# EPICS substitutions: example/example.substitutions
###############################################################################
#
# Positioner template example
#
# $Revision: $
# $Id: $
#
###############################################################################

###############################################################################
#
# Positioner template
#
# The positioner template generates an mbbo record named '$(device):select' that
# is used to select one of n motor positions defined using the position template.
# The output drives the specified motor record '$(motor)'.
#
# interface:
# mbbi   '$(device):select' - use to select the required motor position.
#
# substitutions:
# device  - device name
# motor   - the motor record to be driven
#

file ../db/positioner.template
{
pattern { device, motor }
        { BL18I-DI-PHDGN-01, BL18I-DI-PHDGN-01:MTR }
}

###############################################################################
#
# Position template
# The position template adds '$(device):pos$(idx)' and '$(device):name$(idx)'
# position records to the a positioner template. These specify the motor position
# and the corresponding string name for that position. Up to 16 positions can be
# defined (limited by mbbo record). These records can be changed at run time.
#
# interface
# ao        $(device):pos$(idx)   - use to define the motor position in EGU's at run time
# stringout $(device):name$(idx)  - use to define the name for the position at run time
#
# substitutions:
# device    - device name. This must match the positioner templates $(device) definition.
# pos_name  - the name for the motor position (e.g. a filter name)
# pos_motor - the required motor position in engineering units.
# pos_min   - motor position minimum (in egu's)
# pos_max   - motor position maximum (in egu's)
# pos_egu   - motor position engineering units
# pos_prec  - display precision (PREC) for positions
# idx       - the position suffix (0,1,2...15 corresponding to id)
# id        - one of the EPICS record count prefixes (must be ZR|ON|TW|TH ...FF). (Must be unique for any one positioner)
#

file ../db/position.template
{
pattern { device, pos_name, pos_motor, pos_min, pos_max, pos_egu, pos_prec, idx, id }
        { BL18I-DI-PHDGN-01, filter0, 0, -100, 100, mm, 0, 0, ZR  }
        { BL18I-DI-PHDGN-01, filter1, 20, -100, 100, mm, 0, 1, ON  }
        { BL18I-DI-PHDGN-01, filter2, 50, -100, 100, mm, 0, 2, TW  }
        { BL18I-DI-PHDGN-01, filter3, 95, -100, 100, mm, 0, 3, TH  }
#        { BL18I-DI-PHDGN-01, filter4, 104, -100, 100, mm, 0, 4, FR  }
#        { BL18I-DI-PHDGN-01, filter5, 105, -100, 100, mm, 0, 5, FV  }
#        { BL18I-DI-PHDGN-01, filter6, 106, -100, 100, mm, 0, 6, SX  }
#        { BL18I-DI-PHDGN-01, filter7, 107, -100, 100, mm, 0, 7, SV  }
#        { BL18I-DI-PHDGN-01, filter8, 108, -100, 100, mm, 0, 8, EI  }
#        { BL18I-DI-PHDGN-01, filter9, 109, -100, 100, mm, 0, 9, NI  }
#        { BL18I-DI-PHDGN-01, filter10, 110, -100, 100, mm, 0, 10, TE  }
#        { BL18I-DI-PHDGN-01, filter11, 111, -100, 100, mm, 0, 11, EL  }
#        { BL18I-DI-PHDGN-01, filter12, 112, -100, 100, mm, 0, 12, TV  }
#        { BL18I-DI-PHDGN-01, filter13, 113, -100, 100, mm, 0, 13, TT  }
#        { BL18I-DI-PHDGN-01, filter14, 114, -100, 100, mm, 0, 14, FT  }
#        { BL18I-DI-PHDGN-01, filter15, 115, -100, 100, mm, 0, 15, FF  }
}

###############################################################################

file /home/pjl45/R3.14.7/simulationdev/db/basic_motor.template
{
pattern { P                ,M           ,DESC                 ,DTYP ,DIR ,VELO ,VBAS ,ACCL ,BDST ,BVEL ,BACC ,C ,S ,MRES  ,PREC ,EGU ,DHLM ,DLLM ,INIT }
        { BL18I-DI-PHDGN-01  ,:MTR      ,"Positioner Motor" ,PMAC ,1   ,1000 ,0    ,1    ,0    ,0    ,0    ,0 ,1 ,1     ,5    ,mm  ,100  ,-100 ,""   }
}
